// SIMATIC S7-200 project (STEP 7-Micro/WIN), CPU 221 REL 01.10

ORGANIZATION_BLOCK 主程序:OB1
TITLE=程序注释
BEGIN
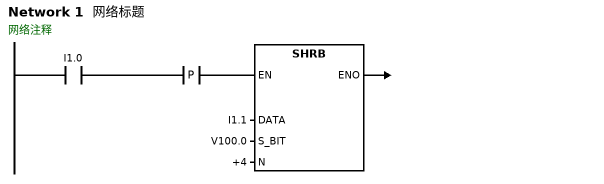
Network 1 // 网络标题
// 网络注释
// (network saved uncompiled; LAD cells follow)
// row 0: c0 -| |- I1.0  c1 -|P|-  c2 [SHRB EN:=power@row0, DATA:=I1.1, S_BIT:=V100.0, N:=+4, ENO=>power]  c3 ->
// row 1: c2 [box]
END_ORGANIZATION_BLOCK
